FUNCTION F_ScalePixel (* Bypass (xScale=FALSE) or scale (xScale=TRUE) one raw pixel value by the DM/SKM factor for u16ObjId. *)
  (* Standard: 61499-2; Description: Copyright (c) 2026 Meisterschulen am Ostbahnhof This program and the accompanying materials are made available under the terms of the Eclipse Public License 2.0 which is available at https://www.eclipse.org/legal/epl-2.0/ SPDX-License-Identifier: EPL-2.0 *)
  (* Version 1.0, 2026-09-05, Franz Höpfinger, Meisterschulen am Ostbahnhof, initial API and implementation and/or initial documentation *)
  PACKAGE isobus::UT::Q::helpers;
  IMPORT isobus::UT::Q::helpers::F_VTScaleFactor;
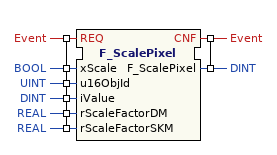
  EVENT_INPUT
    REQ WITH xScale, u16ObjId, iValue, rScaleFactorDM, rScaleFactorSKM;
  END_EVENT
  EVENT_OUTPUT
    CNF WITH F_ScalePixel;
  END_EVENT
  VAR_INPUT
    xScale : BOOL; (* FALSE (default) = bypass, pass iValue through unchanged. TRUE = multiply iValue by the DM/SKM scale factor for u16ObjId. *)
    u16ObjId : UINT; (* Object ID the pixel value belongs to - decides DM vs SKM factor, see F_VTScaleFactor *)
    iValue : DINT; (* Raw pixel value (caller converts its native INT/UINT/USINT field to/from DINT) *)
    rScaleFactorDM : REAL;
    rScaleFactorSKM : REAL;
  END_VAR
  VAR_OUTPUT
    F_ScalePixel : DINT;
  END_VAR
  BODY IN ST:
PACKAGE isobus::UT::Q::helpers;

(* Bypass (xScale=FALSE) or scale (xScale=TRUE) one raw pixel value by the DM/SKM factor
 * for u16ObjId. See F_VTScaleFactor for the ID-range decision. *)
FUNCTION F_ScalePixel : DINT

VAR_INPUT
	xScale : BOOL;
	u16ObjId : UINT;
	iValue : DINT;
	rScaleFactorDM : REAL;
	rScaleFactorSKM : REAL;
END_VAR

IF NOT xScale THEN
	F_ScalePixel := iValue;
ELSE
	F_ScalePixel := REAL_TO_DINT(DINT_TO_REAL(iValue) * F_VTScaleFactor(u16ObjId := u16ObjId, rScaleFactorDM := rScaleFactorDM, rScaleFactorSKM := rScaleFactorSKM));
END_IF;

END_FUNCTION
  END_BODY
END_FUNCTION
